{attribute 'qualified_only'}
VAR_GLOBAL
	Achse2_Ref: AXIS_REF;
	Achse1_Ref: AXIS_REF;
END_VAR

(* stored: Version 1.1.0.1, ProductVersion 3.1.4024.4
   GVL GVL: Id {7fa73dd7-168f-45c4-9ad8-58d202e96f31} *)
